// Mitsubishi GX Works2 project: פרויקט- גרסה לאחר בקר   PLC: FX3G

// global labels: Global1
VAR_GLOBAL
  Start_Workday AT X007 : BOOL;
  Stop_Workday AT X005 : BOOL;  (* מתג כיבוי\ חוסר חומר גלם *)
  Start_Stage1 AT X001 : BOOL;  (* מתג התחלת טעמים *)
  Start_Stage2 AT X002 : BOOL;  (* מתג תחילת קירור *)
  Temp_senseor10 AT X003 : BOOL;  (* חיישן טמפרטורה יורד ל10 מעלות *)
  Day_Light AT Y007 : BOOL;  (* נורת יום עבודה פעיל *)
  Stage1_LighT AT Y000 : BOOL;  (* נורת שלב הכנה פעיל *)
  Cooling_Light AT Y002 : BOOL;  (* נורת שלב קירור םעיל *)
  Mix_Light_1 AT Y005 : BOOL;  (* נורת ערבוב 1 מהבהבת *)
  Mix_Light_2 AT Y006 : BOOL;  (* נורת ערבוב 2 מהבהבת *)
  Stock_Raspberry AT D1100 : REAL;  (* מלאי פטל *)
  Stock_Lemon AT D1102 : REAL;  (* מלאי לימון *)
  Stock_Stabilzer AT D1104 : REAL;  (* מלאי חומר מייצב *)
  Stock_GummyBears AT D1106 : REAL;  (* מלאי דובוני גומי *)
  Total_Packages AT D1108 : REAL;  (* ספירת מארזים שיוצרו *)
  Analog_In_Value AT D1110 : REAL;  (* הערך שידגם מהכניסה האנלוגית לקביעת סוג המארז *)
  System_On_Flag AT M0 : BOOL;  (* זוכר שהמערכת דלוקה *)
  Regular_Package AT M1 : BOOL;  (* דגל שזוכר שהוגרל מארז רגיל *)
  Premium_Package AT M2 : BOOL;  (* דגל שזוכר שהוגרל מארז פינוק *)
  G_Analog_Input_1 AT D8280 : INT;
  Scaled_Analog AT D1112 : REAL;
  RASPBERRY_OK AT M11 : BOOL;  (* דגל שזוכר שהוגרל מארז רגיל *)
  LEMON_OK AT M12 : BOOL;  (* נורת ערבוב 1 מהבהבת *)
  StaBILIZER_OK AT M13 : BOOL;  (* נורת שלב הכנה פעיל *)
  GUMMY_OK AT M14 : BOOL;
  StoCK_OK AT M10 : BOOL;  (* עבר את בדיקות המלאי *)
  Premium_Rasberry_OK AT M21 : BOOL;  (* מלאי פירמיום פירות יער *)
  Premium_Stabilizer_OK AT M23 : BOOL;  (* מלאי פירמיום מייצבים *)
  Premium_LEMON_OK AT M22 : BOOL;  (* מלאי פירמיום לימונים *)
  Premium_GUMMY_OK AT M24 : BOOL;  (* מלאי פירמיום גומי *)
  PREMIUM_StoCK_OK AT M20 : BOOL;  (* עבר את בדיקות מלאי הפרימיום *)
  CoNTINUE_PROCESS AT M30 : BOOL;  (* יש מספיק מלאים להמשך התהליך *)
  SUBTRACTION_DONE AT M40 : BOOL;  (* מניעת הסרה כפולה *)
  Cooling_active AT M50 : BOOL;  (* קירור פעיל *)
  MixING_ACTIVE AT M60 : BOOL;  (* נורת ערבוב 1 מהבהבת *)
  PRODUCT_COUNTER AT D1108 : INT;
  SM412 AT M8013 : BOOL;
  Analog_OUT_VALUE AT D1110 : REAL;  (* הערך שידגם מהכניסה האנלוגית לקביעת סוג המארז *)
  ANALOG_OUTPUT AT D8282 : INT;
  ANALAOG_OUT_INT AT D1116 : INT;
  INIT_RASPBERRY AT D1116 : REAL;
  INIT_STABILIZER AT D1118 : REAL;
  INIT_GUMMYBEARS AT D1120 : REAL;
  INIT_LEMON AT D1122 : REAL;
END_VAR

// task Task_01 (event TRUE, interval 0, priority 31): POU_01

PROGRAM POU_01
VAR
  TON_1 : TON;
  TON_2 : TON;
  TON_3 : TON;
  COUNT_DONE : BOOL;
END_VAR
(* structured ladder/FBD written out as ST: instructions are called as NAME(EN, inputs, outputs); _pN, _eN, _tN stand for wires *)
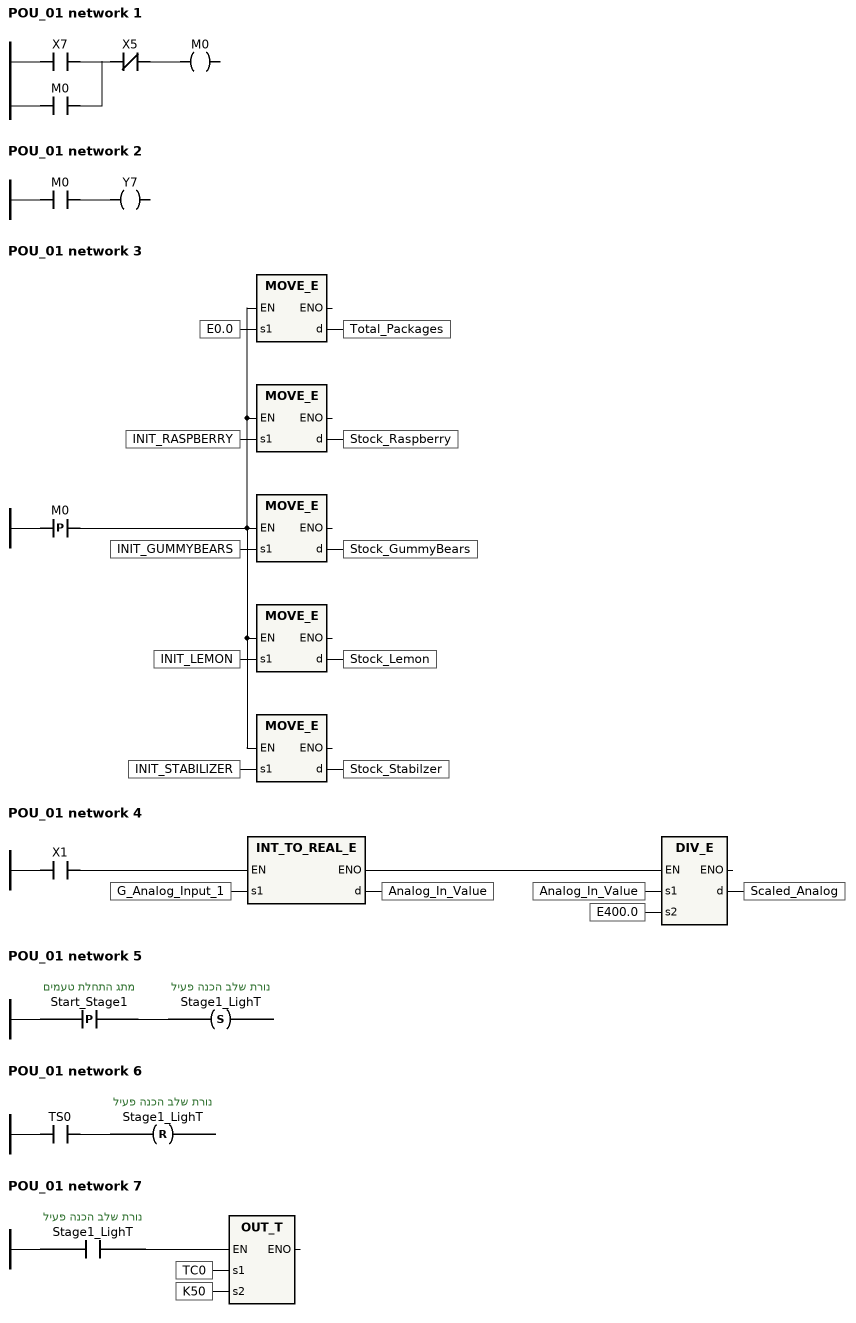
(* network 1 *)
M0 := (X7 OR M0) AND NOT X5;
(* network 2 *)
Y7 := M0;
(* network 3 *)
_p1 := LDP(TRUE, M0);
MOVE_E(_p1, E0.0, Total_Packages);
MOVE_E(_p1, INIT_RASPBERRY, Stock_Raspberry);
MOVE_E(_p1, INIT_GUMMYBEARS, Stock_GummyBears);
MOVE_E(_p1, INIT_LEMON, Stock_Lemon);
MOVE_E(_p1, INIT_STABILIZER, Stock_Stabilzer);
(* network 4 *)
_e1 := INT_TO_REAL_E(X1, G_Analog_Input_1, Analog_In_Value);
DIV_E(_e1, Analog_In_Value, E400.0, Scaled_Analog);
(* network 5 *)
SET(LDP(TRUE, Start_Stage1), Stage1_LighT);
(* network 6 *)
RST(TS0, Stage1_LighT);
(* network 7 *)
OUT_T(Stage1_LighT, TC0, K50);
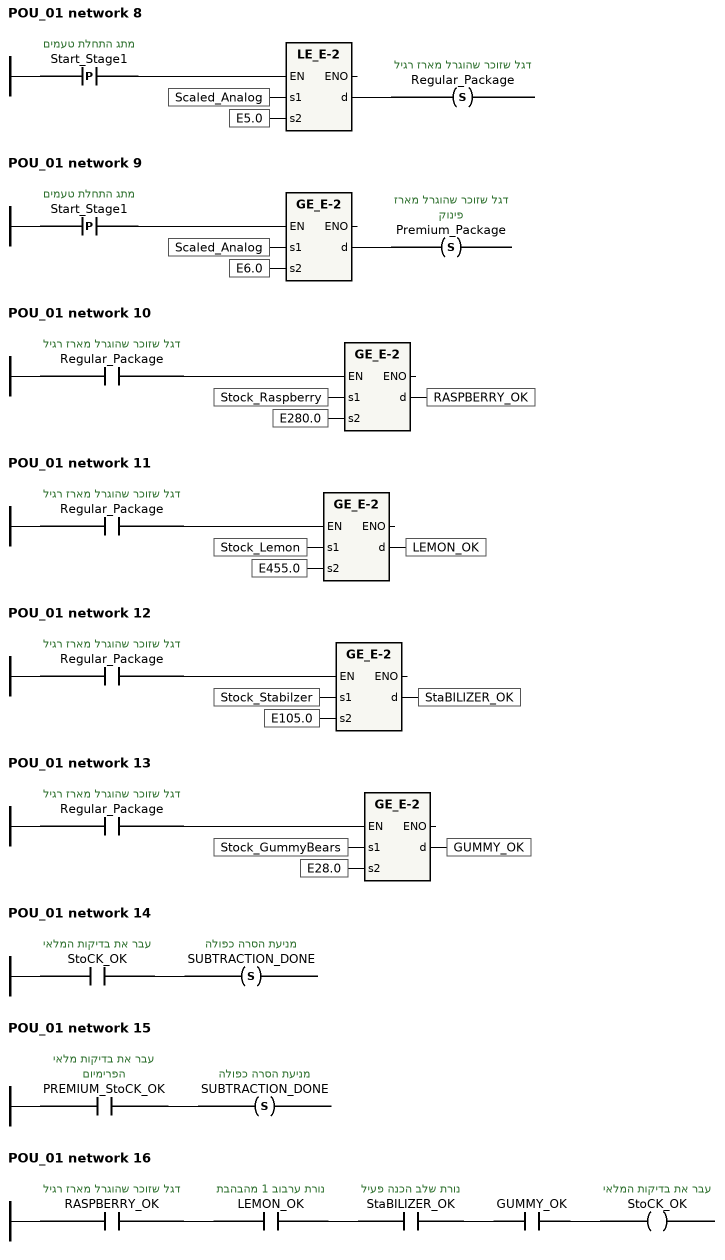
(* network 8 *)
LE_E(LDP(TRUE, Start_Stage1), Scaled_Analog, E5.0, _t1);
SET(_t1, Regular_Package);
(* network 9 *)
GE_E(LDP(TRUE, Start_Stage1), Scaled_Analog, E6.0, _t1);
SET(_t1, Premium_Package);
(* network 10 *)
GE_E(Regular_Package, Stock_Raspberry, E280.0, RASPBERRY_OK);
(* network 11 *)
GE_E(Regular_Package, Stock_Lemon, E455.0, LEMON_OK);
(* network 12 *)
GE_E(Regular_Package, Stock_Stabilzer, E105.0, StaBILIZER_OK);
(* network 13 *)
GE_E(Regular_Package, Stock_GummyBears, E28.0, GUMMY_OK);
(* network 14 *)
SET(StoCK_OK, SUBTRACTION_DONE);
(* network 15 *)
SET(PREMIUM_StoCK_OK, SUBTRACTION_DONE);
(* network 16 *)
StoCK_OK := RASPBERRY_OK AND LEMON_OK AND StaBILIZER_OK AND GUMMY_OK;
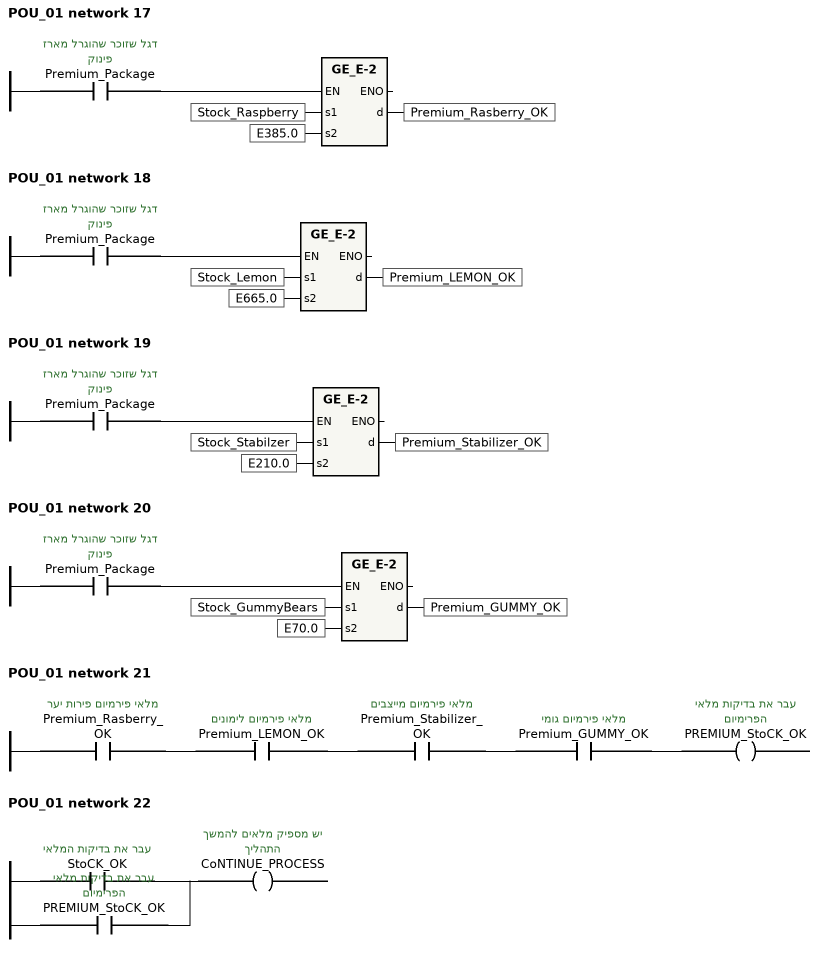
(* network 17 *)
GE_E(Premium_Package, Stock_Raspberry, E385.0, Premium_Rasberry_OK);
(* network 18 *)
GE_E(Premium_Package, Stock_Lemon, E665.0, Premium_LEMON_OK);
(* network 19 *)
GE_E(Premium_Package, Stock_Stabilzer, E210.0, Premium_Stabilizer_OK);
(* network 20 *)
GE_E(Premium_Package, Stock_GummyBears, E70.0, Premium_GUMMY_OK);
(* network 21 *)
PREMIUM_StoCK_OK := Premium_Rasberry_OK AND Premium_LEMON_OK AND Premium_Stabilizer_OK AND Premium_GUMMY_OK;
(* network 22 *)
CoNTINUE_PROCESS := StoCK_OK OR PREMIUM_StoCK_OK;
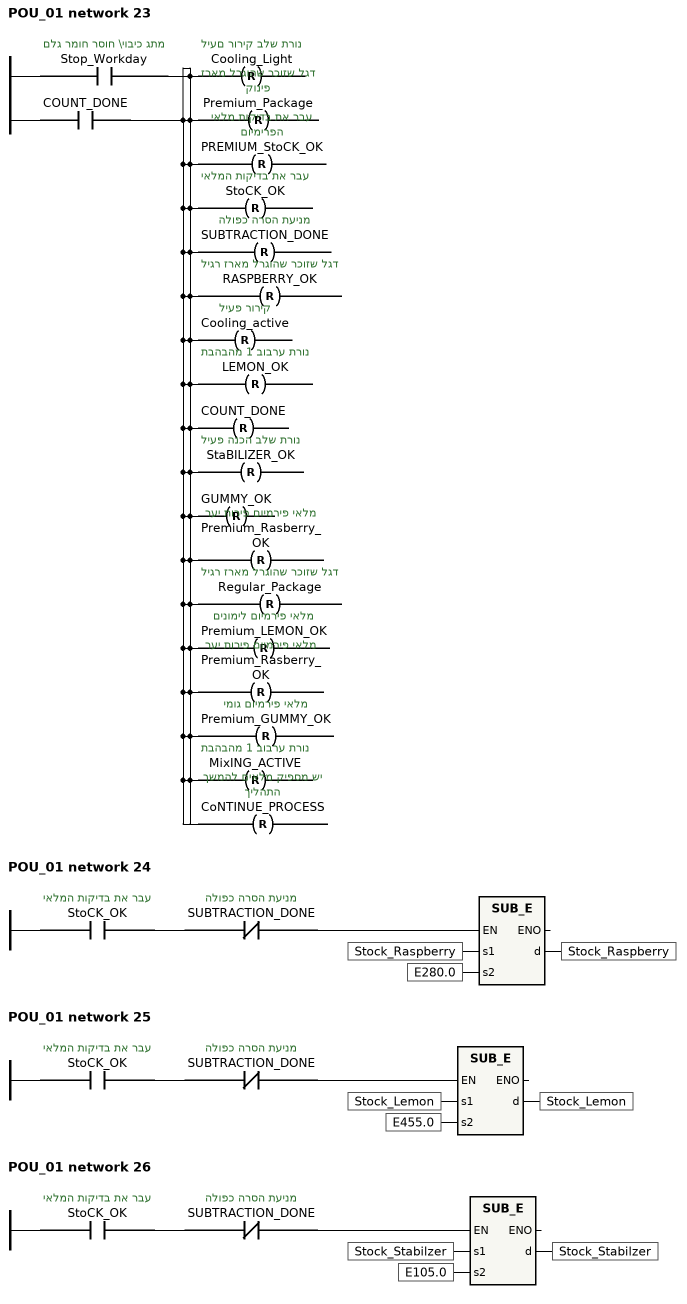
(* network 23 *)
_p1 := Stop_Workday OR COUNT_DONE;
RST(_p1, Cooling_Light);
RST(_p1, Premium_Package);
RST(_p1, PREMIUM_StoCK_OK);
RST(_p1, StoCK_OK);
RST(_p1, SUBTRACTION_DONE);
RST(_p1, RASPBERRY_OK);
RST(_p1, Cooling_active);
RST(_p1, LEMON_OK);
RST(_p1, COUNT_DONE);
RST(_p1, StaBILIZER_OK);
RST(_p1, GUMMY_OK);
RST(_p1, Premium_Rasberry_OK);
RST(_p1, Regular_Package);
RST(_p1, Premium_LEMON_OK);
RST(_p1, Premium_Rasberry_OK);
RST(_p1, Premium_GUMMY_OK);
RST(_p1, MixING_ACTIVE);
RST(_p1, CoNTINUE_PROCESS);
(* network 24 *)
SUB_E(StoCK_OK AND NOT SUBTRACTION_DONE, Stock_Raspberry, E280.0, Stock_Raspberry);
(* network 25 *)
SUB_E(StoCK_OK AND NOT SUBTRACTION_DONE, Stock_Lemon, E455.0, Stock_Lemon);
(* network 26 *)
SUB_E(StoCK_OK AND NOT SUBTRACTION_DONE, Stock_Stabilzer, E105.0, Stock_Stabilzer);
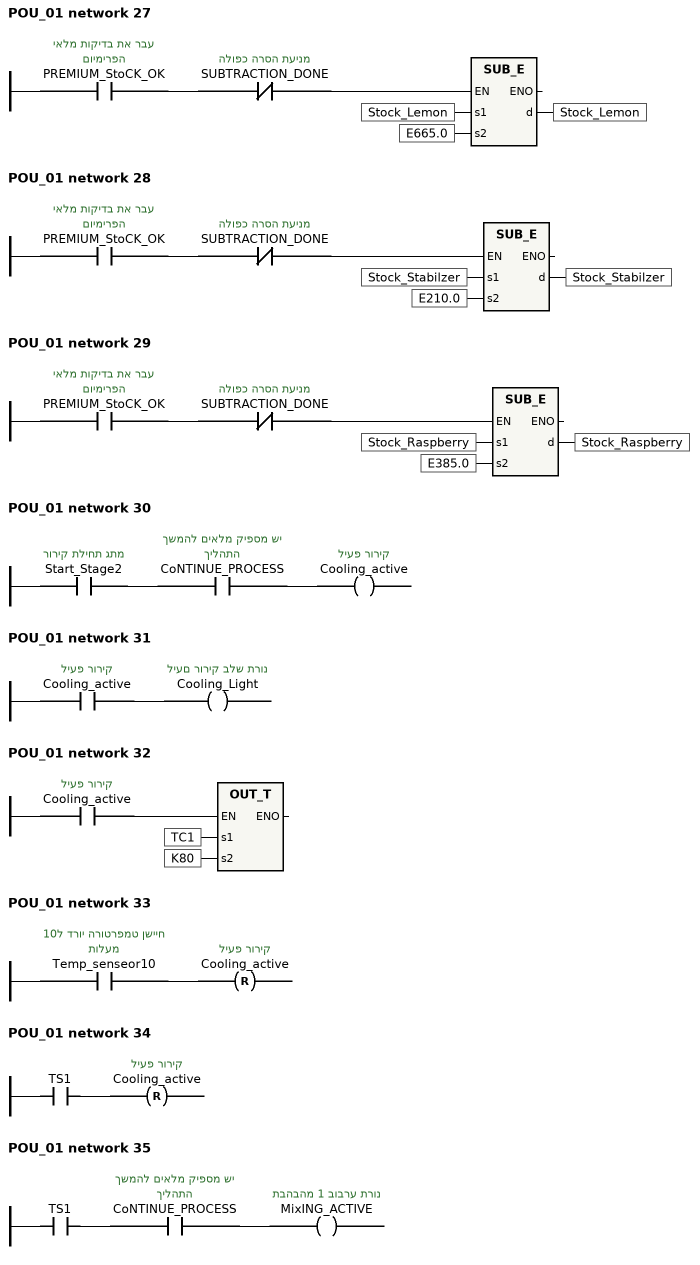
(* network 27 *)
SUB_E(PREMIUM_StoCK_OK AND NOT SUBTRACTION_DONE, Stock_Lemon, E665.0, Stock_Lemon);
(* network 28 *)
SUB_E(PREMIUM_StoCK_OK AND NOT SUBTRACTION_DONE, Stock_Stabilzer, E210.0, Stock_Stabilzer);
(* network 29 *)
SUB_E(PREMIUM_StoCK_OK AND NOT SUBTRACTION_DONE, Stock_Raspberry, E385.0, Stock_Raspberry);
(* network 30 *)
Cooling_active := Start_Stage2 AND CoNTINUE_PROCESS;
(* network 31 *)
Cooling_Light := Cooling_active;
(* network 32 *)
OUT_T(Cooling_active, TC1, K80);
(* network 33 *)
RST(Temp_senseor10, Cooling_active);
(* network 34 *)
RST(TS1, Cooling_active);
(* network 35 *)
MixING_ACTIVE := TS1 AND CoNTINUE_PROCESS;
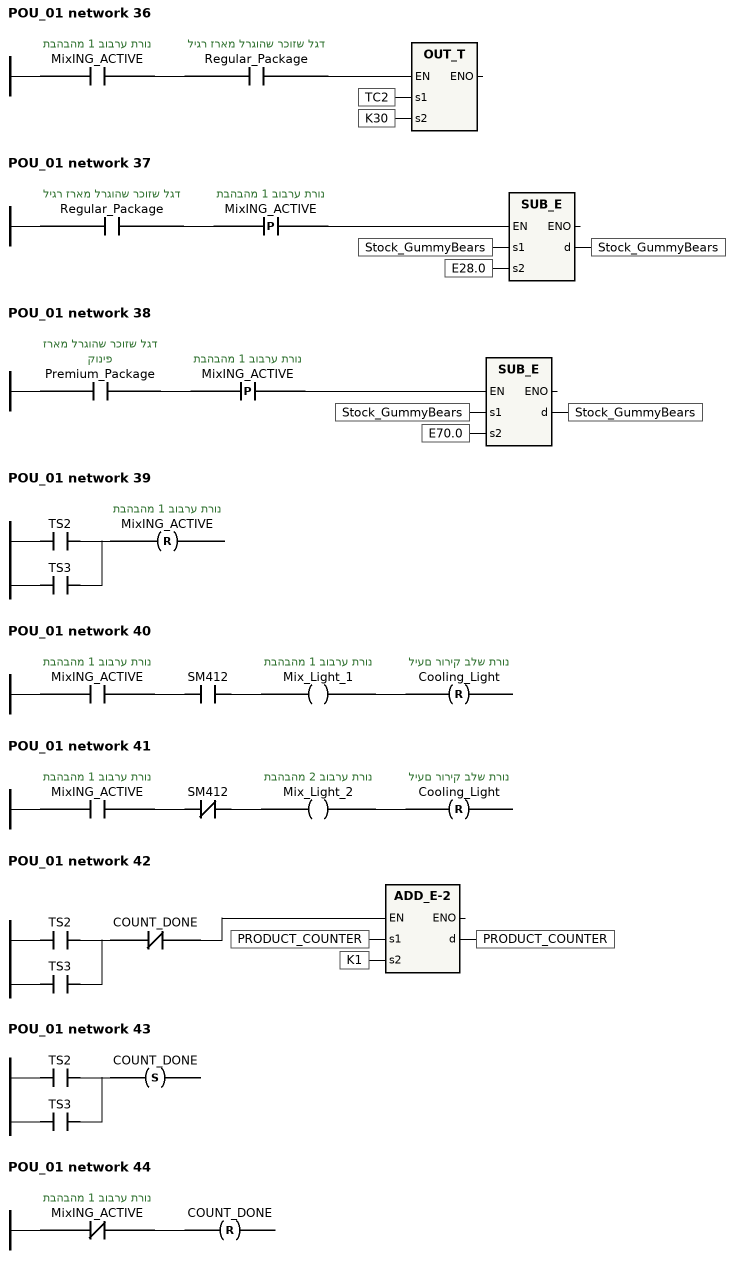
(* network 36 *)
OUT_T(MixING_ACTIVE AND Regular_Package, TC2, K30);
(* network 37 *)
SUB_E(Regular_Package AND LDP(TRUE, MixING_ACTIVE), Stock_GummyBears, E28.0, Stock_GummyBears);
(* network 38 *)
SUB_E(Premium_Package AND LDP(TRUE, MixING_ACTIVE), Stock_GummyBears, E70.0, Stock_GummyBears);
(* network 39 *)
RST(TS2 OR TS3, MixING_ACTIVE);
(* network 40 *)
_p1 := MixING_ACTIVE AND SM412;
Mix_Light_1 := _p1;
RST(_p1, Cooling_Light);
(* network 41 *)
_p1 := MixING_ACTIVE AND NOT SM412;
Mix_Light_2 := _p1;
RST(_p1, Cooling_Light);
(* network 42 *)
ADD_E((TS2 OR TS3) AND NOT COUNT_DONE, PRODUCT_COUNTER, K1, PRODUCT_COUNTER);
(* network 43 *)
SET(TS2 OR TS3, COUNT_DONE);
(* network 44 *)
RST(NOT MixING_ACTIVE, COUNT_DONE);
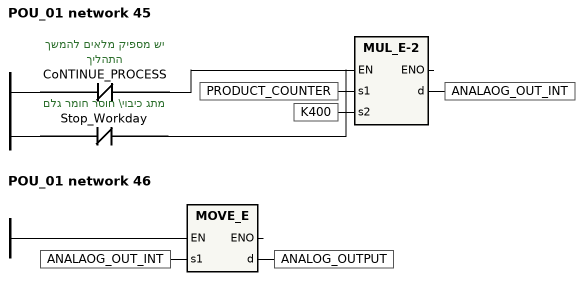
(* network 45 *)
MUL_E((NOT CoNTINUE_PROCESS) OR (NOT Stop_Workday), PRODUCT_COUNTER, K400, ANALAOG_OUT_INT);
(* network 46 *)
MOVE_E(TRUE, ANALAOG_OUT_INT, ANALOG_OUTPUT);
END_PROGRAM
